{attribute 'strict'}
TYPE E_MachineCtrlStateAbort :
(
	MACHINE_STATE_ABORTING_TABLE					:= 0,	(*  *)
	MACHINE_STATE_ABORTING_ROBOT_CYCLE_STOP			:= 10,	(*  *)
	MACHINE_STATE_ABORTING_DONE						:= 200	(*  *)
);
END_TYPE

(* stored: Version 1.1.0.1, ProductVersion 3.1.4024.9
   DUT E_MachineCtrlStateAbort: Id {d5ac7684-2254-418c-a115-fb375f618847} *)
